// TIA Portal V19 export
DATA_BLOCK "AckProcessAndPbAlarms"   // DB3
{ S7_Optimized_Access := 'TRUE' }
AUTHOR : FLA
FAMILY : UHT
VERSION : 1.0
// stored: AutoNumber false, MemoryReserve 0
   VAR
      "A" : Array[1..96] of Bool;
   END_VAR
BEGIN
   // "A"[1] : A01_TankInProcess
   // "A"[2] : A02_TankNotClean
   // "A"[3] : A03_NoInstrumentAir
   // "A"[4] : A04_NoSteam
   // "A"[5] : A05_DrainIsActive
   // "A"[6] : A06_CipFillerStarted
   // "A"[7] : A07_CipUnitOccupied
   // "A"[8] : A08_NotReadyForCip
   // "A"[9] : A09_NoProcessActive
   // "A"[10] : A10_AllreadyInStopPhase
   // "A"[11] : A11_TankIsBeingFilled
   // "A"[12] : A12_NotReadyForTotalStop
   // "A"[13] : A13_DrainTankNotAllowed
   // "A"[14] : A14_CipOnTankStared
   // "A"[15] : A15_ChainWashSelected
   // "A"[16] : A16_NoCipProgramSelected
   // "A"[17] : A17_ContinueDosingSelect
   // "A"[18] : A18
   // "A"[19] : A19
   // "A"[20] : A20
   // "A"[21] : A21
   // "A"[22] : A22
   // "A"[23] : A23
   // "A"[24] : A24
   // "A"[25] : A25
   // "A"[26] : A26
   // "A"[27] : A27
   // "A"[28] : A28
   // "A"[29] : A29
   // "A"[30] : A30
   // "A"[31] : A31
   // "A"[32] : A32
   // "A"[33] : A33_TT0176TooLow
   // "A"[34] : A34_TT0160TooLow
   // "A"[35] : A35_TT0163TooLow
   // "A"[36] : A36_TT0178TooLow
   // "A"[37] : A37_TT0176Low
   // "A"[38] : A38_TT0178Low
   // "A"[39] : A39_TankReadyforProd
   // "A"[40] : A40_LyedosingTooLong
   // "A"[41] : A41_AcidDosingTooLong
   // "A"[42] : A42_DrainTheTank
   // "A"[43] : A43_WaitingForCipUnit
   // "A"[44] : A44_FillPressureTooLow
   // "A"[45] : A45_FillingPressureLow
   // "A"[46] : A46_LyeContainerEmpty
   // "A"[47] : A47_AcidContainerEmpty
   // "A"[48] : A48_TankEmpty
   // "A"[49] : A49_TankFull
   // "A"[50] : A50_SiemensBatteryLow
   // "A"[51] : A51_NoWater
   // "A"[52] : A52_ProdAtFillingMash
   // "A"[53] : A53_FillerNotReadyForCip
   // "A"[54] : A54_NoInstrumentAir
   // "A"[55] : A55_NoSteam
   // "A"[56] : A56
   // "A"[57] : A57_TT0951TooLow
   // "A"[58] : A58_TT0951Low
   // "A"[59] : A59_TT0950TooLow
   // "A"[60] : A60_TT0950Low
   // "A"[61] : A61_Hamba_Valve_Fault
   // "A"[62] : A62_Hamba_Barrier_low
   // "A"[63] : dx7_6_Spare
   // "A"[64] : dx7_7_Spare
   // "A"[65] : dx8_0_Spare
   // "A"[66] : dx8_1_Spare
   // "A"[67] : dx8_2_Spare
   // "A"[68] : dx8_3_Spare
   // "A"[69] : dx8_4_Spare
   // "A"[70] : dx8_5_Spare
   // "A"[71] : dx8_6_Spare
   // "A"[72] : dx8_7_Spare
   // "A"[73] : dx9_0_Spare
   // "A"[74] : dx9_1_Spare
   // "A"[75] : dx9_2_Spare
   // "A"[76] : dx9_3_Spare
   // "A"[77] : dx9_4_Spare
   // "A"[78] : dx9_5_Spare
   // "A"[79] : dx9_6_Spare
   // "A"[80] : dx9_7_Spare
   // "A"[81] : dx10_0_Spare
   // "A"[82] : dx10_1_Spare
   // "A"[83] : dx10_2_Spare
   // "A"[84] : dx10_3_Spare
   // "A"[85] : dx10_4_Spare
   // "A"[86] : dx10_5_Spare
   // "A"[87] : dx10_6_Spare
   // "A"[88] : dx10_7_Spare
   // "A"[89] : dx11_0_Spare
   // "A"[90] : dx11_1_Spare
   // "A"[91] : dx11_2_Spare
   // "A"[92] : dx11_3_Spare
   // "A"[93] : dx11_4_Spare
   // "A"[94] : dx11_5_Spare
   // "A"[95] : dx11_6_Spare
   // "A"[96] : dx11_7_Spare
END_DATA_BLOCK
